// TIA Portal V18 export
FUNCTION_BLOCK "Block_2_1"   // FB2, LAD
{ S7_Optimized_Access := 'TRUE' }
VERSION : 0.1
// stored: AutoNumber true, IsIECCheckEnabled false, IsRetainMemResEnabled false, MemoryReserve 100, SetENOAutomatically false, UDAEnableTagReadback false
   VAR_INPUT
      qwe : Bool;
   END_VAR
   VAR
      SEQ01_InterruptState : Bool;
      SEQ01_SingleStep_Bit : Bool;
      ST04_OS01_Condition : Bool;
      ST04_OS01 : Bool;
      ST14 : Bool;
      ST14_OS01 : Bool;
      ST13_OS01 : Bool;
      ST14_OS01_Condition : Bool;
   END_VAR
   VAR_TEMP
      ST04 : Bool;
   END_VAR
BEGIN

REGION Network 1: @@@[ST14] Wait_for_Seq_Over: Within Step
   // @@@<Wait_for_Seq_Over> Active
   // Jump from <Wait_for_Work_Complete_ACK> by ST13_OS01
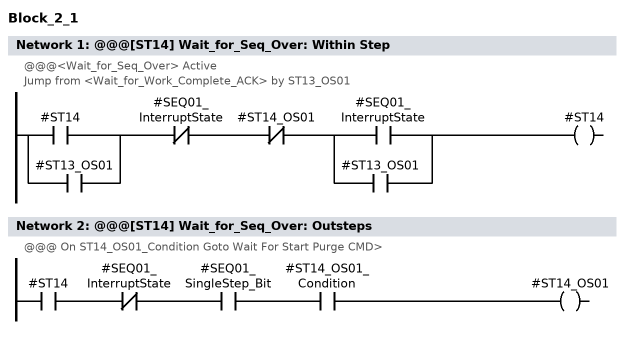
   RUNG wire#powerrail
      Contact( #ST14 )
      wire#w1
      I_Contact( #SEQ01_InterruptState )
      I_Contact( #ST14_OS01 )
      wire#w2
      Contact( #SEQ01_InterruptState )
      wire#w3
      Coil( #ST14 )
   END_RUNG
   RUNG wire#powerrail
      Contact( #ST13_OS01 )
   END_RUNG wire#w1
   RUNG wire#w2
      Contact( #ST13_OS01 )
   END_RUNG wire#w3
   // the same network as SCL:
   #ST14 := (#ST14 OR #ST13_OS01) AND NOT #SEQ01_InterruptState AND NOT #ST14_OS01 AND (#SEQ01_InterruptState OR #ST13_OS01);
END_REGION

REGION Network 2: @@@[ST14] Wait_for_Seq_Over: Outsteps
   // @@@ On ST14_OS01_Condition Goto Wait For Start Purge CMD>
   RUNG wire#powerrail
      Contact( #ST14 )
      I_Contact( #SEQ01_InterruptState )
      Contact( #SEQ01_SingleStep_Bit )
      Contact( #ST14_OS01_Condition )
      Coil( #ST14_OS01 )
   END_RUNG
   // the same network as SCL:
   #ST14_OS01 := #ST14 AND NOT #SEQ01_InterruptState AND #SEQ01_SingleStep_Bit AND #ST14_OS01_Condition;
END_REGION
END_FUNCTION_BLOCK
